FUNCTION_BLOCK L4_FMS205_F2SeqPrep_SFC EXTENDS L1_ControllerBase_SFC
// Girar 8 veces el plato para determinar qué tipo de tapa hay en cada sector del plato
VAR_INPUT
	cnF2_Preparar	: BOOL;
	Siguiente		: BOOL := FALSE;
	Medid			: REFERENCE TO L3_MedidorTapa;
	Induc		 	: REFERENCE TO L3_CaptadorInductivo;
	Fotoe			: REFERENCE TO L3_DetectorFotoelectrico;
	Plato			: REFERENCE TO L3_PlatoDivisor;
END_VAR

VAR_OUTPUT
	Seguir 	 		: BOOL;	
	Giros 			: INT := 0;
END_VAR

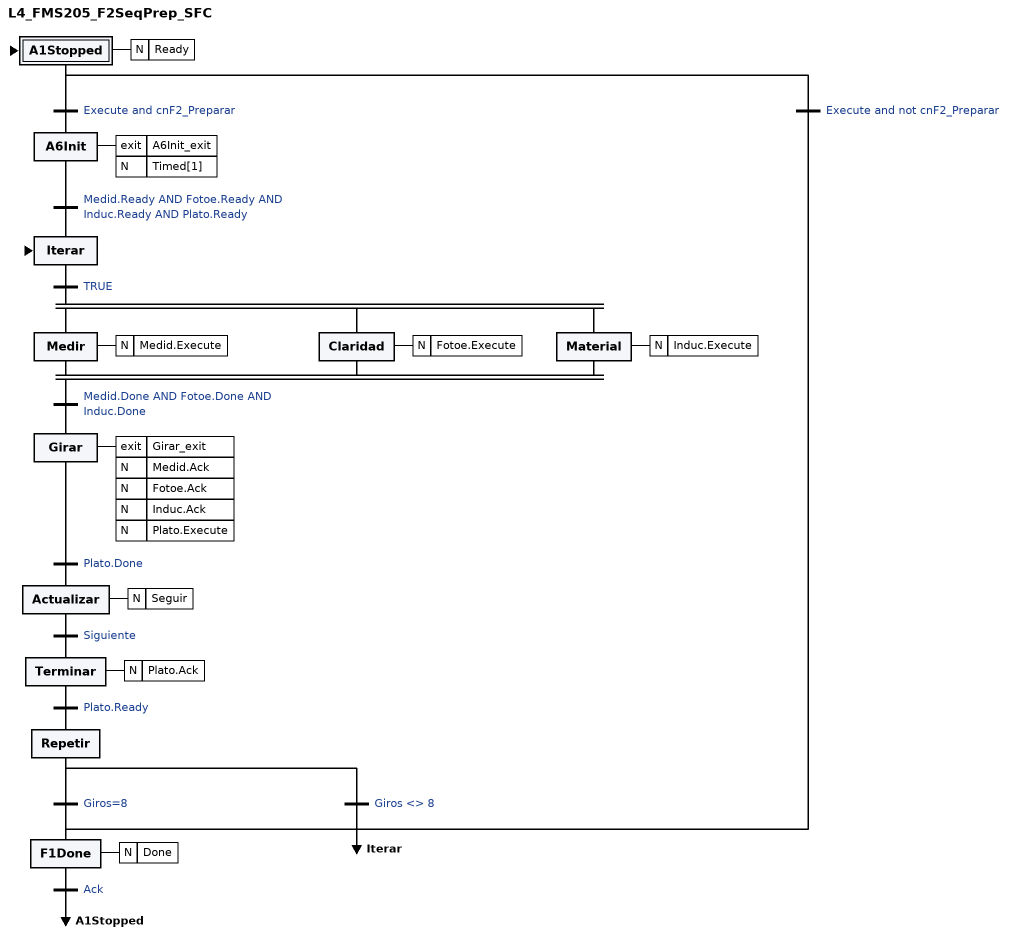
INITIAL_STEP A1Stopped:
    Ready(N);
END_STEP
TRANSITION FROM A1Stopped TO A6Init
    := Execute and cnF2_Preparar;
END_TRANSITION
STEP A6Init:
    A6Init_exit(P0);  // exit action
    Timed[1](N);
END_STEP
TRANSITION FROM A6Init TO Iterar
    := Medid.Ready AND Fotoe.Ready AND Induc.Ready AND Plato.Ready;
END_TRANSITION
STEP Iterar:
END_STEP
TRANSITION FROM Iterar TO (Medir, Claridad, Material)
    := TRUE;
END_TRANSITION
STEP Medir:
    Medid.Execute(N);
END_STEP
STEP Claridad:
    Fotoe.Execute(N);
END_STEP
STEP Material:
    Induc.Execute(N);
END_STEP
TRANSITION FROM (Medir, Claridad, Material) TO Girar
    := Medid.Done AND Fotoe.Done AND Induc.Done;
END_TRANSITION
STEP Girar:
    Girar_exit(P0);  // exit action
    Medid.Ack(N);
    Fotoe.Ack(N);
    Induc.Ack(N);
    Plato.Execute(N);
END_STEP
TRANSITION FROM Girar TO Actualizar
    := Plato.Done;
END_TRANSITION
STEP Actualizar:
    Seguir(N);
END_STEP
TRANSITION FROM Actualizar TO Terminar
    := Siguiente;
END_TRANSITION
STEP Terminar:
    Plato.Ack(N);
END_STEP
TRANSITION FROM Terminar TO Repetir
    := Plato.Ready;
END_TRANSITION
STEP Repetir:
END_STEP
TRANSITION FROM Repetir TO F1Done
    := Giros=8;
END_TRANSITION
TRANSITION FROM Repetir TO Iterar
    := Giros <> 8;
END_TRANSITION
TRANSITION FROM A1Stopped TO F1Done
    := Execute and not cnF2_Preparar;
END_TRANSITION
STEP F1Done:
    Done(N);
END_STEP
TRANSITION FROM F1Done TO A1Stopped
    := Ack;
END_TRANSITION

ACTION A6Init_exit:
Giros:=0;
END_ACTION

ACTION Girar_exit:
Giros:=Giros+1;
END_ACTION

END_FUNCTION_BLOCK

(* stored: Version 1.1.0.1, ProductVersion 3.1.4024.11
   POU L4_FMS205_F2SeqPrep_SFC: Id {306e8fb2-9473-4dd1-ac8a-7196779de084}, SpecialFunc None
   Action A6Init_exit: Id {e1190fd2-b61b-4572-abcd-f44d34d42ffc}
   Action Girar_exit: Id {50a4a834-adbe-40c6-b72d-eb4caaf0978f} *)
